INTERFACE I_AsynchronousCommandBusyState

METHOD PUBLIC SetAborting
VAR_INPUT
END_VAR
END_METHOD

METHOD PUBLIC SetDone
VAR_INPUT
END_VAR
END_METHOD

METHOD PUBLIC SetError
VAR_INPUT
	ErrorId : UDINT;
END_VAR
END_METHOD

END_INTERFACE

(* stored: Version 1.1.0.1, ProductVersion 3.1.4024.11
   Itf I_AsynchronousCommandBusyState: Id {ac32b9d1-66c3-4455-9f40-dadf7044247c}
   Method SetAborting: Id {e0e67b54-8972-43b1-a296-2dc05d87b1ea}
   Method SetDone: Id {47c318cd-5679-4ddc-8cf8-61abad24bb2a}
   Method SetError: Id {35548a66-2856-4f6f-8555-895f708279db} *)
